(* IEC 61131-3 sources: Industry-PLC-LLM/data/PLCBEAD_repo/PLCBEAD_PLCEmbed-main/PLC-BEAD/Source/GEB/K_TO_C, 1 file *)

(* ---- K_TO_C.ST ---- *)
FUNCTION K_TO_C:REAL

	VAR_INPUT
		KELVIN :	REAL;
	END_VAR

	K_TO_C := KELVIN + 273.15;

END_FUNCTION

PROGRAM program0
	VAR
		KELVIN : REAL;
		OUT : REAL;
	END_VAR

	OUT := K_TO_C(KELVIN);
END_PROGRAM
